(* CoDeSys 2.3 export: TANALOGINPUT.EXP *)

(* Data type *)
TYPE tAnalogInput : REAL;
END_TYPE
